TYPE T_MODBUS_STAT EXTENDS T_RS_COMM_STAT:
STRUCT
	DeviceReply: 		ARRAY [0..300] OF BYTE;
	nValue:				DINT;	// Value read from the device
END_STRUCT
END_TYPE

(* stored: Version 1.1.0.1, ProductVersion 3.1.4022.16
   DUT T_MODBUS_STAT: Id {e5d4f5de-a3b4-4218-a867-4a0b5180985c} *)
